FUNCTION_BLOCK FB_EMAG_Y
VAR_INPUT
	bCN_Demand : BOOL;
	bError_Connection : BOOL;
END_VAR
VAR_OUTPUT
END_VAR
VAR
	//I/O-Links
	Mode_IN AT %I* : BOOL;
	CoolingUnitOperational_IN AT %I* : BOOL;
	ConnectionStatus_IN AT %I* : BOOL;

END_VAR

bCN_Demand := CoolingUnitOperational_IN AND ConnectionStatus_IN;
bError_Connection := NOT ConnectionStatus_IN;

END_FUNCTION_BLOCK

(* stored: Version 1.1.0.1, ProductVersion 3.1.4024.10
   POU FB_EMAG_Y: Id {a864166e-4288-4090-96e6-3b67cc736d1a}, SpecialFunc None *)
